PROGRAM MAIN
VAR
END_VAR

END_PROGRAM

(* stored: Version 1.1.0.1
   POU MAIN: Id {46b766b9-540e-481f-8de5-0dfb8ff2cc4d} *)
